screen "statistic" 800x480, template "Main"
   Rectangle "Rectangle_33" at 0,128 size 732x281
      Visibility <- "Vis_reset_stat"
   TextField "Text field_68" at 197,132 size 338x58; Text 'Новая партия.'
      Visibility <- "Vis_reset_stat"
   Button "Button_15" at 135,324 size 196x75; TextOff 'Продолжить'
      on Click: SetBit("T3V3W3_DB_Reset_statistic"); ResetBit("Vis_reset_stat")
      Visibility <- "Vis_reset_stat"
   Button "Button_6" at 391,323 size 196x75; TextOff 'Отмена'
      on Click: ResetBit("Vis_reset_stat")
      Visibility <- "Vis_reset_stat"
   TextField "Text field_69" at 200,186 size 333x46; Text 'Название партии:'
      Visibility <- "Vis_reset_stat"
   TextField "Text field_70" at 118,295 size 498x28; Text 'В партии может быть максимум 3000 коробок!'
      Visibility <- "Vis_reset_stat"
   IOField "I/O field_57" at 60,232 size 613x48; FormatPattern ?????????????????????????
      ProcessValue <- "T3V3W3_DB_LocalVar_name_part"
      Visibility <- "Vis_reset_stat"
   Button "Button_5" at 14,415 size 211x58; TextOff 'Обзор'
      on Click: ActivateScreen("Root screen", 0); SetTag("main_screens", 0)
      Appearance <- "main_screens"
   Button "Button_14" at 264,415 size 211x58; TextOff 'Вес'
      on Click: ActivateScreen("weight", 0); SetTag("main_screens", 1)
      Appearance <- "main_screens"
   Button "Button_7" at 513,415 size 211x58; TextOff 'Статистика'
      on Click: ActivateScreen("statistic", 0); SetTag("main_screens", 2); SetTag("stat_view", 0)
      Appearance <- "main_screens"
   Button "Button_8" at 150,363 size 211x46; TextOff 'Данные'
      on Click: ActivateScreen("statistic", 0); SetTag("stat_view", 0)
      Appearance <- "stat_view"
   Button "Button_9" at 372,363 size 211x46; TextOff 'Память'
      on Click: ActivateScreen("Memory", 0); SetTag("stat_view", 1)
      Appearance <- "stat_view"
   IOField "I/O field_1" at 122,58 size 57x22; FormatPattern 99.99
      ProcessValue <- "Statistic_DB_move_stat_Instance_box_weight{1}"
   TextField "Text field_1" at 122,0 size 231x23; Text 'Вес по коробкам в партии:'
   IOField "I/O field_2" at 153,29 size 47x22; FormatPattern 9999
      ProcessValue <- "b_1"
   TextField "Text field_2" at 122,29 size 43x23; Text '№'
   TextField "Text field_3" at 181,58 size 43x23; Text 'кг'
   IOField "I/O field_3" at 122,126 size 57x22; FormatPattern 99.99
      ProcessValue <- "Statistic_DB_move_stat_Instance_box_weight{6}"
   IOField "I/O field_4" at 153,96 size 47x22; FormatPattern 9999
      ProcessValue <- "b_6"
   TextField "Text field_4" at 122,96 size 43x23; Text '№'
   TextField "Text field_5" at 181,126 size 43x23; Text 'кг'
   IOField "I/O field_5" at 122,193 size 57x22; FormatPattern 99.99
      ProcessValue <- "Statistic_DB_move_stat_Instance_box_weight{11}"
   IOField "I/O field_6" at 153,164 size 47x22; FormatPattern 9999
      ProcessValue <- "b_11"
   TextField "Text field_6" at 122,164 size 43x23; Text '№'
   TextField "Text field_7" at 181,193 size 43x23; Text 'кг'
   IOField "I/O field_7" at 122,261 size 57x22; FormatPattern 99.99
      ProcessValue <- "Statistic_DB_move_stat_Instance_box_weight{16}"
   IOField "I/O field_8" at 153,231 size 47x22; FormatPattern 9999
      ProcessValue <- "b_16"
   TextField "Text field_8" at 122,231 size 43x23; Text '№'
   TextField "Text field_9" at 181,261 size 43x23; Text 'кг'
   IOField "I/O field_9" at 122,329 size 57x22; FormatPattern 99.99
      ProcessValue <- "Statistic_DB_move_stat_Instance_box_weight{21}"
   IOField "I/O field_10" at 153,299 size 47x22; FormatPattern 9999
      ProcessValue <- "b_21"
   TextField "Text field_10" at 122,299 size 43x23; Text '№'
   TextField "Text field_11" at 181,329 size 43x23; Text 'кг'
   IOField "I/O field_11" at 232,58 size 57x22; FormatPattern 99.99
      ProcessValue <- "Statistic_DB_move_stat_Instance_box_weight{2}"
   IOField "I/O field_12" at 263,29 size 47x22; FormatPattern 9999
      ProcessValue <- "b_2"
   TextField "Text field_12" at 232,29 size 43x23; Text '№'
   TextField "Text field_13" at 291,58 size 43x23; Text 'кг'
   IOField "I/O field_13" at 232,126 size 57x22; FormatPattern 99.99
      ProcessValue <- "Statistic_DB_move_stat_Instance_box_weight{7}"
   IOField "I/O field_14" at 263,96 size 47x22; FormatPattern 9999
      ProcessValue <- "b_7"
   TextField "Text field_14" at 232,96 size 43x23; Text '№'
   TextField "Text field_15" at 291,126 size 43x23; Text 'кг'
   IOField "I/O field_15" at 232,193 size 57x22; FormatPattern 99.99
      ProcessValue <- "Statistic_DB_move_stat_Instance_box_weight{12}"
   IOField "I/O field_16" at 263,164 size 47x22; FormatPattern 9999
      ProcessValue <- "b_12"
   TextField "Text field_16" at 232,164 size 43x23; Text '№'
   TextField "Text field_17" at 291,193 size 43x23; Text 'кг'
   IOField "I/O field_17" at 232,261 size 57x22; FormatPattern 99.99
      ProcessValue <- "Statistic_DB_move_stat_Instance_box_weight{17}"
   IOField "I/O field_18" at 263,231 size 47x22; FormatPattern 9999
      ProcessValue <- "b_17"
   TextField "Text field_18" at 232,231 size 43x23; Text '№'
   TextField "Text field_19" at 291,261 size 43x23; Text 'кг'
   IOField "I/O field_19" at 232,329 size 57x22; FormatPattern 99.99
      ProcessValue <- "Statistic_DB_move_stat_Instance_box_weight{22}"
   IOField "I/O field_20" at 263,299 size 47x22; FormatPattern 9999
      ProcessValue <- "b_22"
   TextField "Text field_20" at 232,299 size 43x23; Text '№'
   TextField "Text field_21" at 291,329 size 43x23; Text 'кг'
   IOField "I/O field_21" at 342,58 size 57x22; FormatPattern 99.99
      ProcessValue <- "Statistic_DB_move_stat_Instance_box_weight{3}"
   IOField "I/O field_22" at 373,29 size 47x22; FormatPattern 9999
      ProcessValue <- "b_3"
   TextField "Text field_22" at 342,29 size 43x23; Text '№'
   TextField "Text field_23" at 401,58 size 43x23; Text 'кг'
   IOField "I/O field_23" at 342,126 size 57x22; FormatPattern 99.99
      ProcessValue <- "Statistic_DB_move_stat_Instance_box_weight{8}"
   IOField "I/O field_24" at 373,96 size 47x22; FormatPattern 9999
      ProcessValue <- "b_8"
   TextField "Text field_24" at 342,96 size 43x23; Text '№'
   TextField "Text field_25" at 401,126 size 43x23; Text 'кг'
   IOField "I/O field_25" at 342,193 size 57x22; FormatPattern 99.99
      ProcessValue <- "Statistic_DB_move_stat_Instance_box_weight{13}"
   IOField "I/O field_26" at 373,164 size 47x22; FormatPattern 9999
      ProcessValue <- "b_13"
   TextField "Text field_26" at 342,164 size 43x23; Text '№'
   TextField "Text field_27" at 401,193 size 43x23; Text 'кг'
   IOField "I/O field_27" at 342,261 size 57x22; FormatPattern 99.99
      ProcessValue <- "Statistic_DB_move_stat_Instance_box_weight{18}"
   IOField "I/O field_28" at 373,231 size 47x22; FormatPattern 9999
      ProcessValue <- "b_18"
   TextField "Text field_28" at 342,231 size 43x23; Text '№'
   TextField "Text field_29" at 401,261 size 43x23; Text 'кг'
   IOField "I/O field_29" at 342,329 size 57x22; FormatPattern 99.99
      ProcessValue <- "Statistic_DB_move_stat_Instance_box_weight{23}"
   IOField "I/O field_30" at 373,299 size 47x22; FormatPattern 9999
      ProcessValue <- "b_23"
   TextField "Text field_30" at 342,299 size 43x23; Text '№'
   TextField "Text field_31" at 401,329 size 43x23; Text 'кг'
   IOField "I/O field_31" at 452,58 size 57x22; FormatPattern 99.99
      ProcessValue <- "Statistic_DB_move_stat_Instance_box_weight{4}"
   IOField "I/O field_32" at 483,29 size 47x22; FormatPattern 9999
      ProcessValue <- "b_4"
   TextField "Text field_32" at 452,29 size 43x23; Text '№'
   TextField "Text field_33" at 511,58 size 43x23; Text 'кг'
   IOField "I/O field_33" at 452,126 size 57x22; FormatPattern 99.99
      ProcessValue <- "Statistic_DB_move_stat_Instance_box_weight{9}"
   IOField "I/O field_34" at 483,96 size 47x22; FormatPattern 9999
      ProcessValue <- "b_9"
   TextField "Text field_34" at 452,96 size 43x23; Text '№'
   TextField "Text field_35" at 511,126 size 43x23; Text 'кг'
   IOField "I/O field_35" at 452,193 size 57x22; FormatPattern 99.99
      ProcessValue <- "Statistic_DB_move_stat_Instance_box_weight{14}"
   IOField "I/O field_36" at 483,164 size 47x22; FormatPattern 9999
      ProcessValue <- "b_14"
   TextField "Text field_36" at 452,164 size 43x23; Text '№'
   TextField "Text field_37" at 511,193 size 43x23; Text 'кг'
   IOField "I/O field_37" at 452,261 size 57x22; FormatPattern 99.99
      ProcessValue <- "Statistic_DB_move_stat_Instance_box_weight{19}"
   IOField "I/O field_38" at 483,231 size 47x22; FormatPattern 9999
      ProcessValue <- "b_19"
   TextField "Text field_38" at 452,231 size 43x23; Text '№'
   TextField "Text field_39" at 511,261 size 43x23; Text 'кг'
   IOField "I/O field_39" at 452,329 size 57x22; FormatPattern 99.99
      ProcessValue <- "Statistic_DB_move_stat_Instance_box_weight{24}"
   IOField "I/O field_40" at 483,299 size 47x22; FormatPattern 9999
      ProcessValue <- "b_24"
   TextField "Text field_40" at 452,299 size 43x23; Text '№'
   TextField "Text field_41" at 511,329 size 43x23; Text 'кг'
   IOField "I/O field_41" at 562,58 size 57x22; FormatPattern 99.99
      ProcessValue <- "Statistic_DB_move_stat_Instance_box_weight{5}"
   IOField "I/O field_42" at 593,29 size 47x22; FormatPattern 9999
      ProcessValue <- "b_5"
   TextField "Text field_42" at 562,29 size 43x23; Text '№'
   TextField "Text field_43" at 621,58 size 43x23; Text 'кг'
   IOField "I/O field_43" at 562,126 size 57x22; FormatPattern 99.99
      ProcessValue <- "Statistic_DB_move_stat_Instance_box_weight{10}"
   IOField "I/O field_44" at 593,96 size 47x22; FormatPattern 9999
      ProcessValue <- "b_10"
   TextField "Text field_44" at 562,96 size 43x23; Text '№'
   TextField "Text field_45" at 621,126 size 43x23; Text 'кг'
   IOField "I/O field_45" at 562,193 size 57x22; FormatPattern 99.99
      ProcessValue <- "Statistic_DB_move_stat_Instance_box_weight{15}"
   IOField "I/O field_46" at 593,164 size 47x22; FormatPattern 9999
      ProcessValue <- "b_15"
   TextField "Text field_46" at 562,164 size 43x23; Text '№'
   TextField "Text field_47" at 621,193 size 43x23; Text 'кг'
   IOField "I/O field_47" at 562,261 size 57x22; FormatPattern 99.99
      ProcessValue <- "Statistic_DB_move_stat_Instance_box_weight{20}"
   IOField "I/O field_48" at 593,231 size 47x22; FormatPattern 9999
      ProcessValue <- "b_20"
   TextField "Text field_48" at 562,231 size 43x23; Text '№'
   TextField "Text field_49" at 621,261 size 43x23; Text 'кг'
   IOField "I/O field_49" at 562,329 size 57x22; FormatPattern 99.99
      ProcessValue <- "Statistic_DB_move_stat_Instance_box_weight{25}"
   IOField "I/O field_50" at 593,299 size 47x22; FormatPattern 9999
      ProcessValue <- "b_25"
   TextField "Text field_50" at 562,299 size 43x23; Text '№'
   TextField "Text field_51" at 621,329 size 43x23; Text 'кг'
   GraphicView "Graphic view_1" at 664,24 size 57x50; Picture "u_grey"
   GraphicView "Graphic view_2" at 662,309 size 57x50; Picture "nope"
   TextField "Text field_52" at 22,21 size 72x23; Text 'Партия:'
   TextField "Text field_54" at 5,60 size 82x23; Text 'Коробок:'
   IOField "I/O field_52" at 36,78 size 47x22; FormatPattern 9999
      ProcessValue <- "T3V3W3_DB_Statistic_Count"
   TextField "Text field_55" at 81,78 size 43x23; Text 'шт'
   TextField "Text field_56" at 5,94 size 77x42; Text 'Средний вес:'
   IOField "I/O field_53" at 32,131 size 77x22; FormatPattern 99.99
      ProcessValue <- "T3V3W3_DB_Statistic_Mid_weight"
   TextField "Text field_57" at 81,131 size 43x23; Text 'кг'
   Button "Button_1" at 663,25 size 57x50; TextOff 'Text'
      on Click: SetBit("Statistic_DB_move_stat_Instance_up")
   Button "Button_2" at 663,309 size 57x50; TextOff 'Text'
      on Click: SetBit("Statistic_DB_move_stat_Instance_down")
   TextField "Text field_58" at 22,187 size 72x23; Text 'Партия:'
   TextField "Text field_59" at 17,205 size 82x23; Text 'Прошлая'
   TextField "Text field_60" at 9,228 size 82x23; Text 'Коробок:'
   IOField "I/O field_55" at 40,246 size 47x22; FormatPattern 9999
      ProcessValue <- "T3V3W3_DB_Statistic_Count_old"
   TextField "Text field_61" at 85,246 size 43x23; Text 'шт'
   TextField "Text field_62" at 9,259 size 77x42; Text 'Средний вес:'
   IOField "I/O field_56" at 35,296 size 54x22; FormatPattern 99.99
      ProcessValue <- "T3V3W3_DB_Statistic_Mid_weight_old"
   TextField "Text field_63" at 81,296 size 43x23; Text 'кг'
   TextField "Text field_53" at 6,38 size 104x23; Text 'Актуальная'
   Button "Button_3" at 658,165 size 69x52; TextOff 'Новая партия'
      on Click: SetBit("Vis_reset_stat")
      Visibility <- "Logic_DB_Start_weight"
   TextField "Text field_64" at 5,147 size 87x23; Text 'Общ. вес:'
   IOField "I/O field_51" at 8,165 size 77x22; FormatPattern 99999.9
      ProcessValue <- "T3V3W3_DB_Statistic_Weight"
   TextField "Text field_65" at 80,163 size 43x23; Text 'кг'
   TextField "Text field_66" at 9,313 size 87x23; Text 'Общ. вес:'
   IOField "I/O field_54" at 12,331 size 77x22; FormatPattern 99999.9
      ProcessValue <- "T3V3W3_DB_Statistic_Weight_old"
   TextField "Text field_67" at 84,329 size 43x23; Text 'кг'
   Button "Button_4" at 658,79 size 69x52; TextOff 'В начало'
      on Click: SetBit("Statistic_DB_move_stat_Instance_In_the_beggin")
   IOField "I/O field_58" at 352,1 size 313x22; FormatPattern ?????????????????????????
      ProcessValue <- "T3V3W3_DB_LocalVar_name_part"

Template "Main" 800x480
   Button "Button_1" at 735,5 size 60x60; TextOff 'Text'; PictureOff "home_2"
      on Click: ActivateScreen("Root screen", 0); SetTag("main_screens", 0)
   Button "Button_2" at 735,84 size 60x60; TextOff 'Text'; PictureOff "sett"
      on Click: ActivateScreen("SP", 0); SetTag("Sp_view", 1)
   Button "Button_4" at 735,163 size 60x60; TextOff 'Text'; PictureOff "sett_1"
      on Click: ActivateScreen("Monitor", 0); SetTag("settings", 0)
   Button "Button_5" at 735,242 size 60x60; TextOff 'Text'; PictureOff "home_1"; PictureList "Alarm"
      on Click: ActivateScreen("Alarms", 0)
      ProcessValue <- "Any_Alm"
   Button "Button_6" at 735,321 size 60x60; TextOff 'Text'; PictureOff "back"
      on Click: function_efd93a16()
   Button "Button_7" at 735,401 size 60x60; TextOff 'Text'; PictureOff "reset"
      on Click: SetBit("Reset_All")
   TextField "Template_Text field_1" at 735,63 size 60x15; Text 'F3'
   TextField "Template_Text field_2" at 735,222 size 60x15; Text 'F5'
   TextField "Template_Text field_3" at 735,143 size 60x15; Text 'F4'
   TextField "Template_Text field_4" at 735,300 size 60x15; Text 'F6'
   TextField "Template_Text field_5" at 735,460 size 60x15; Text 'F8'
   TextField "Template_Text field_6" at 735,380 size 60x15; Text 'F7'

screen "1.1_Recalibration" 800x480, template "Template_1"
   TextField "OBJECT_35" at 0,2 size 510x34; Text '1.1.1 Mit Gewichten Nachjustieren / 1.1 Recalibration / 1.1.1 Réétalonnage avec poids étalon / Calibration'
   Button "Exit to Service" at 45,390 size 80x80; TextOn 'Texte / text'; TextOff 'Texte / text'; PictureOff "Exit"
      on Release: ActivateScreen("Monitor", 0); SetTag("WP231PR_DB_CMD_A", 2034)
      on Press: SetTag("WP231PR_DB_s_CMD2_i_CMD_CODE", '2'); SetBit("WP231PR_DB_s_CMD2_bo_CMD_TRIGGER"); SetTag("WP231PR_DB_CMD_B", 0)
   Group "Group" at 700,5 size 95x30; Text 'Service'; PictureList "Signal_grey_yellow"
   Button "Up_to Setup_5_Min_01" at 545,390 size 80x80; TextOn 'Texte / text'; TextOff 'Texte / text'; PictureOff "Left"
      on Release: SetTag("WP231PR_DB_CMD_A", 2034)
      on Press: ActivateScreen("0.0.0_Service_Recalibration", 0); SetTag("WP231PR_DB_CMD_B", 0)
   IOField "OBJECT_301" at 0,41 size 800x90; FormatPattern ????????????????
      ProcessValue <- "WP231PR_DB_DR34_ASCII_DISPLAY"
   Button "OBJECT_28" at 110,133 size 580x70; TextOn 'Texte / text'; TextOff 'Justagegewicht 0 setzen / Set Calibration Weight 0 / Placez le poids étalon 0 / Acknowledge Empty Bin'
      on Press: SetTag("WP231PR_DB_s_CMD2_i_CMD_CODE", '60'); SetBit("WP231PR_DB_s_CMD2_bo_CMD_TRIGGER")
   Button "OBJECT_31" at 110,204 size 580x70; TextOn 'Texte / text'; TextOff 'Justagegewicht 1 setzen / Set Calibration Weight 1 / Placez le poids étalon 1 / Put & Acknowledge Calibration Weight'
      on Press: SetTag("WP231PR_DB_s_CMD2_i_CMD_CODE", '61'); SetBit("WP231PR_DB_s_CMD2_bo_CMD_TRIGGER")
   Button "OBJECT_3" at 110,276 size 580x70; TextOn 'Texte / text'; TextOff 'Justagegewicht 2 setzen (optional) / Set Calibration Weight 2 (optional) / Placez le poids étalon 2 (option) / Put & Acknowledge Calibration Weight'
      on Press: SetTag("WP231PR_DB_s_CMD2_i_CMD_CODE", '62'); SetBit("WP231PR_DB_s_CMD2_bo_CMD_TRIGGER")
   Button "Schaltfläche_1" at 670,390 size 80x80; TextOn 'Texte'; TextOff 'Texte'; PictureOff "Q_Mark"
      on Press: SetBit("S1_SHOW_HELP")
   TextField "OBJECT_4" at 210,352 size 207x32; Text 'Aktuelle Digits ADC: / Current ADC digits: / Valeur CAN / Error occurred'
      Visibility <- "S1_SHOW_HELP"
   IOField "I/O field_5" at 442,351 size 136x32; FormatPattern 9999999999
      ProcessValue <- "WP231PR_DB_DR31_DIGITS_FILTERED"
      Visibility <- "S1_SHOW_HELP"
   GraphicIOField "OBJECT_19" at 765,5 size 30x30; PictureList "Signal_grey_yellow"
      ProcessValue <- "WP231PR_DB_s_IO_DATA_SCALE_STATUS_2_SERVICE_MODE"
   TextField "OBJECT_37" at 700,7 size 57x25; Text 'Service / Error occurred'
   Rectangle "Rechteck_1" at 0,131 size 799x348
      Visibility <- "S1_SHOW_HELP"
   TextField "OBJECT_2" at 73,165 size 334x47; Text 'Justagegewicht 0: / Calibration weight 0: / Poids étalon 0: / Calibration'
      Visibility <- "S1_SHOW_HELP"
   TextField "OBJECT_1" at 73,230 size 334x47; Text 'Justagegewicht 1: / Calibration weight 1: / Poids étalon 1: / Calibration'
      Visibility <- "S1_SHOW_HELP"
   IOField "I/O field_1" at 415,230 size 166x47; FormatPattern 99999.99
      ProcessValue <- "WP231PR_DB_DR03_CALIB_WEIGHT_1"
      Visibility <- "S1_SHOW_HELP"
   IOField "I/O field_2" at 571,230 size 134x47; FormatPattern ????
      ProcessValue <- "WP231PR_DB_DR03_WEIGHT_UNIT"
      Visibility <- "S1_SHOW_HELP"
   IOField "I/O field_3" at 415,165 size 166x47; FormatPattern 99999.99
      ProcessValue <- "WP231PR_DB_DR03_CALIB_WEIGHT_0"
      Visibility <- "S1_SHOW_HELP"
   IOField "I/O field_4" at 571,165 size 134x47; FormatPattern ????
      ProcessValue <- "WP231PR_DB_DR03_WEIGHT_UNIT"
      Visibility <- "S1_SHOW_HELP"
   TextField "OBJECT_5" at 73,300 size 334x47; Text 'Justagegewicht 2: / Calibration weight 2: / Poids étalon 2: / Calibration'
      Visibility <- "S1_SHOW_HELP"
   IOField "I/O field_6" at 415,300 size 166x47; FormatPattern 99999.99
      ProcessValue <- "WP231PR_DB_DR03_CALIB_WEIGHT_2"
      Visibility <- "S1_SHOW_HELP"
   IOField "I/O field_7" at 571,300 size 134x47; FormatPattern ????
      ProcessValue <- "WP231PR_DB_DR03_WEIGHT_UNIT"
      Visibility <- "S1_SHOW_HELP"
   Button "Schaltfläche_2" at 642,420 size 150x50; TextOn 'Texte'; TextOff 'OK'
      on Press: ResetBit("S1_SHOW_HELP")
      Visibility <- "S1_SHOW_HELP"

screen "1.2.1_Quick_Start_1" 800x480, template "Template_1"
   TextField "OBJECT_33" at 0,0 size 440x34; Text '1.2.1 Quick Start 1 von 5 / 1.2.1 Quick Start 1 of 5 / 1.2.1 Mise en service rapide 1/5 / Setup 1/3'
   Button "Exit to Service" at 45,390 size 80x80; TextOn 'Texte / text'; TextOff 'Texte / text'; PictureOff "Exit"
      on Release: ActivateScreen("Monitor", 0)
      on Press: SetTag("WP231PR_DB_s_CMD2_i_CMD_CODE", '2'); SetBit("WP231PR_DB_s_CMD2_bo_CMD_TRIGGER")
   Button "Factory settings" at 110,112 size 580x90; TextOn 'Texte / text'; TextOff '"Quick Start" mit bestehenden Einstellungen / Run "Quick Start" with existing settings / Démarrage rapide avec les paramètres actuels / Acknowledge Empty Bin'
      on Release: ActivateScreen("1.2.2_Quick_Start_2", 0)
      on Press: SetTag("WP231PR_DB_s_CMD2_i_CMD_CODE", '2003'); SetBit("WP231PR_DB_s_CMD2_bo_CMD_TRIGGER")
   Group "Group" at 700,5 size 95x30; Text 'Service'; PictureList "Signal_grey_yellow"
   Button "Factory settings_1" at 110,237 size 580x90; TextOn 'Texte / text'; TextOff '"Quick Start" mit Werkseinstellungen / Run "Quick Start" with factory default settings / Démarrage rapide avec les paramètres usine / Acknowledge Empty Bin'
      on Release: ActivateScreen("1.2.2_Quick_Start_2", 0); SetTag("WP231PR_DB_s_CMD2_i_CMD_CODE", '2003'); SetBit("WP231PR_DB_s_CMD2_bo_CMD_TRIGGER")
      on Press: SetTag("WP231PR_DB_s_CMD1_i_CMD_CODE", 12); SetBit("WP231PR_DB_s_CMD1_bo_CMD_TRIGGER")
   Button "Schaltfläche_1" at 360,390 size 80x80; TextOn 'Texte'; TextOff 'Texte'; PictureOff "Q_Mark"
      on Press: SetBit("S1_SHOW_HELP")
   GraphicIOField "OBJECT_19" at 765,5 size 30x30; PictureList "Signal_grey_yellow"
      ProcessValue <- "WP231PR_DB_s_IO_DATA_SCALE_STATUS_2_SERVICE_MODE"
   TextField "OBJECT_37" at 700,7 size 57x25; Text 'Service / Error occurred'
   TextField "Textfeld_1" at 0,57 size 800x422; Text '"Quick Start" ermöglicht eine schnelle Basis-Inbetriebnahme der Waage. Es besteht die Möglichkeit die Waage mit oder ohne Justagegewichte zu justieren. "Quick Start" kann mit den bestehenden Waagenparametern, als auch mit geladenen Werkseinstellungen durchgeführt werden. "Quick Start" allows a fast and easy basic commissioning of the scale. It is possible to calibrate the scale with or without calibration weights. You can enter the "Quick Start" procedure with loaded factory settings or with maintaining the scale settings. Le démarrage rapide pour une mise en service en quelques minutes'
      Visibility <- "S1_SHOW_HELP"
   Button "Schaltfläche_2" at 643,423 size 150x50; TextOn 'Texte'; TextOff 'OK'
      on Press: ResetBit("S1_SHOW_HELP")
      Visibility <- "S1_SHOW_HELP"

screen "1.2.2_Quick_Start_2" 800x480, template "Template_1"
   TextField "OBJECT_33" at 0,0 size 440x34; Text '1.2.2 Quick Start 2 von 5 / 1.2.2 Quick Start 2 of 5 / 1.2.2 Mise en service rapide 2/5 / Setup 1/3'
   Button "Exit to Service" at 45,390 size 80x80; TextOn 'Texte / text'; TextOff 'Texte / text'; PictureOff "Exit"
      on Release: ActivateScreen("Monitor", 0)
      on Press: SetTag("WP231PR_DB_s_CMD2_i_CMD_CODE", '2'); SetBit("WP231PR_DB_s_CMD2_bo_CMD_TRIGGER")
   Group "Group" at 700,5 size 95x30; Text 'Service'; PictureList "Signal_grey_yellow"
   TextField "OBJECT_306" at 234,90 size 179x29; Text 'Waagenname / Scale Name / Nom de la balance / Scale name'
   IOField "OBJECT_307" at 420,84 size 172x40; HelpText 'Name der Waage (Produkt, Anlagenteil o.Ä.) / Nom de la balance'; FormatPattern ????????????
      ProcessValue <- "WP231PR_DB_DR03_SCALE_NAME"
   TextField "OBJECT_7" at 258,141 size 151x29; Text 'Gewichtseinheit / Weight unit / Unité poids / Weight Unit'
   IOField "OBJECT_28" at 420,134 size 172x40; HelpText 'Gewichtseinheit (z.B. g, kg oder t) / Unité poids (par ex. g, kg ou t)'; FormatPattern ????
      ProcessValue <- "WP231PR_DB_DR03_WEIGHT_UNIT"
   TextField "OBJECT_9" at 129,285 size 283x29; Text 'Minimaler Wägebereich (in d) / Minimum weight (in d) / Poids min (en d) / Weight Unit'
   TextField "OBJECT_10" at 159,330 size 254x29; Text 'Maximaler Wägebereich / Maximum weight / Plage maximale de pesage / Weight Unit'
   TextField "OBJECT_11" at 252,237 size 159x29; Text 'Ziffernschritt (d) / Resolution / Résolution (d) / Weight Unit'
   IOField "OBJECT_29" at 420,279 size 172x40; HelpText 'Bei geeichten Waagen mind. 20 x Ziffernschritt d. Bei nicht eichpflichtigen Waagen kann der minimale Wägebereich mit 0 definiert werden. / 20 x d pour usage certifié, sinon pas de limitation (0 par exemple)'; FormatPattern 999
      ProcessValue <- "WP231PR_DB_DR03_MIN_WEIGHT_D"
   IOField "OBJECT_12" at 420,325 size 173x40; HelpText 'Maximales Gewicht auf der Waage. Bei geeichten Waagen bitte entsprechende Einschränkungen beachten! / Poids max. sur la balance'; FormatPattern 9999999.9999
      ProcessValue <- "WP231PR_DB_DR03_MAX_WEIGHT"
   IOField "OBJECT_13" at 420,230 size 172x40; HelpText 'Ziffernschritt der Waage. Ist die Gewichts einheit "kg" bedeutet ein Ziffernschritt von 0,1 dass die Waage in 0,1kg Schritten auflöst. / Résolution de la balance. Avec un unité de poids de 1kg, la résolution de 0,1 signifie 0,1kg'; FormatPattern 9999.9999
      ProcessValue <- "WP231PR_DB_DR03_RESOLUTION_D"
   IOField "I/O field_2" at 596,325 size 60x40; FormatPattern ????
      ProcessValue <- "WP231PR_DB_DR03_WEIGHT_UNIT"
   TextField "Textfeld_1" at 609,283 size 18x29; Text 'x'
   Group "Group_1" at 607,242 size 62x59
   Button "Down to Setup_5_Min_03" at 690,390 size 80x80; TextOn 'Texte / text'; TextOff 'Texte / text'; PictureOff "Right"
      on Release: ActivateScreen("1.2.3_Quick_Start_3", 0)
   Button "Up_to Setup_5_Min_01" at 545,390 size 80x80; TextOn 'Texte / text'; TextOff 'Texte / text'; PictureOff "Left"
      on Release: ActivateScreen("1.2.1_Quick_Start_1", 0)
   TextField "OBJECT_6" at 8,188 size 403x29; Text 'Brutto-Kennung ("B" oder "G") / Indicator for Gross ("B" or "G") / Abréviation pour le poids brut ("B" ou "G") / Weight Unit'
   SymbolicIOField "Symbolic I/O field_1" at 421,187 size 172x31; TextOn '1'; TextOff '0'; TextList "003030_LETTER_FOR_GROSS_WEIGHT"
      ProcessValue <- "WP231PR_DB_DR03_LETTER_GROSS_WEIGHT_2"
   Button "Down to Setup_5_Min_1" at 360,390 size 80x80; TextOn 'Texte / text'; TextOff 'Texte / text'; PictureOff "Save"
      on Press: SetTag("WP231PR_DB_s_CMD2_i_CMD_CODE", '4003'); SetBit("WP231PR_DB_s_CMD2_bo_CMD_TRIGGER")
   GraphicIOField "OBJECT_19" at 765,5 size 30x30; PictureList "Signal_grey_yellow"
      ProcessValue <- "WP231PR_DB_s_IO_DATA_SCALE_STATUS_2_SIMULATION_MODE"
   TextField "OBJECT_37" at 700,7 size 57x25; Text 'Service / Error occurred'

screen "1.2.3_Quick_Start_3" 800x480, template "Template_1"
   TextField "OBJECT_35" at 0,0 size 440x34; Text '1.2.3 Quick Start 3 von 5 / 1.2.3 Quick Start 3 of 5 / 1.2.3 Mise en service rapide 3/5 / Quick Setup'
   Button "Exit to Service" at 45,390 size 80x80; TextOn 'Texte / text'; TextOff 'Texte / text'; PictureOff "Exit"
      on Release: ActivateScreen("Monitor", 0)
      on Press: SetTag("WP231PR_DB_s_CMD2_i_CMD_CODE", '2'); SetBit("WP231PR_DB_s_CMD2_bo_CMD_TRIGGER")
   TextField "OBJECT_38" at 34,80 size 762x32; Text 'Soll die Waage mit oder ohne Gewichte justiert werden? / Do you want to calibrate the scale with or without weights? / Calibration avec ou sans poids étalon? / For Quick Setup the scale must be empty'
   Button "Up_to Setup_5_Min_01" at 545,390 size 80x80; TextOn 'Texte / text'; TextOff 'Texte / text'; PictureOff "Left"
      on Release: ActivateScreen("1.2.2_Quick_Start_2", 0)
   Group "Group" at 700,5 size 95x30; Text 'Service'; PictureList "Signal_grey_yellow"
   Button "Factory settings" at 110,138 size 580x90; TextOn 'Texte / text'; TextOff 'Mit Gewichten justieren / Calibrate With Weights / Etalonner avec des poids étalons / Acknowledge Empty Bin'
      on Release: ActivateScreen("1.2.4_Quick_Start_Manual_Calibration_1", 0)
   Button "Factory settings_1" at 110,263 size 580x90; TextOn 'Texte / text'; TextOff 'Ohne Gewichte justieren (automatisch) Calibrate without weights (automatic) Calibration sans poids étalon Acknowledge Empty Bin'
      on Release: ActivateScreen("1.2.6_Quick_Start_4", 0)
      on Press: SetTag("WP231PR_DB_s_CMD2_i_CMD_CODE", '2010'); SetBit("WP231PR_DB_s_CMD2_bo_CMD_TRIGGER")
   Softkey "Softkey_F4" at -140,-147 size 0x0
      on KeyDown: ActivateScreen("1.2.6_Quick_Start_4", 0)
   GraphicIOField "OBJECT_19" at 765,5 size 30x30; PictureList "Signal_grey_yellow"
      ProcessValue <- "WP231PR_DB_s_IO_DATA_SCALE_STATUS_2_SERVICE_MODE"
   TextField "OBJECT_37" at 700,7 size 57x25; Text 'Service / Error occurred'
   TextField "Textfeld_1" at 0,57 size 800x422; Text 'Justage mit Gewichten: Es müssen mindestens 5% der Nennlast der Waage als Justagegewicht zur Verfügung stehen. Beispiel: 3 x 2t Wägezellen = 6t Nennlast --> Die Waage muss mit mindestens 300kg (5% von 6t) justiert werden. Wird der Justagepunkt 2 ebenfalls genutzt, muss dieser wiederum mindestens 300kg vom Justagepunkt 1 entfernt sein. Automatische Justage: Es sind keine Justagegewichte notwendig. Die Wägezellendaten müssen zur Verfügung stehen. Mechanische Einflüsse werden nicht berücksichtigt! Etalonnage avec un poids étalon. Au min 5% de la charge nominale des pesons'
      Visibility <- "S1_SHOW_HELP"
   Button "Schaltfläche_2" at 643,423 size 150x50; TextOn 'Texte'; TextOff 'OK'
      on Press: ResetBit("S1_SHOW_HELP")
      Visibility <- "S1_SHOW_HELP"

screen "1.2.4_Quick_Start_Manual_Calibration_1" 800x480, template "Template_1"
   TextField "OBJECT_33" at 0,0 size 630x34; Text '1.2.4 Quick Start - Justagegewichte 4 von 5 / 1.2.4 Quick Start - Calibration Weights 4 of 5 / 1.2.4 Mise en service rapide poids étalon 4/5 / Setup 1/3'
   TextField "OBJECT_306" at 157,135 size 206x32; Text 'Justagegewicht 0 / Calibration weight 0 / Poids étalon 0 / Scale name'
   Button "OBJECT_34" at 670,390 size 80x80; TextOn 'Texte / text'; TextOff 'Texte / text'; PictureOff "Right"
      on Release: ActivateScreen("1.2.5_Quick_Start_Manual_Calibration_2", 0); SetTag("WP231PR_DB_CMD_A", 2034)
      on Press: SetTag("WP231PR_DB_CMD_B", 2031)
   IOField "OBJECT_307" at 373,126 size 300x50; HelpText 'Falls die Waage zum Zeitpunkt der Justage nicht leer ist, kann das bekannte Gewicht in der Waage als "Justagegewicht 0" vorgegeben werden. / If the scale is not empty before adjusting, the known material weight in the scale can be defined as "Calibration weight 0". / Si pour l'étalonnage la balance n'est pas vide, il est possible d'utiliser le poids actuel comme poids étalon'; FormatPattern 999999.999
      ProcessValue <- "WP231PR_DB_DR03_CALIB_WEIGHT_0"
   TextField "OBJECT_7" at 158,192 size 206x32; Text 'Justagegewicht 1 / Calibration weight 1 / Poids étalon 1 / Weight Unit'
   IOField "OBJECT_28" at 373,182 size 300x50; HelpText 'Das "Justagegewicht 1" muss mindestens 5% der Nennlast der Waage entsprechen! / Le poids étalon doit être supérieur à 5% de la charge max des pesons'; FormatPattern 999999.999
      ProcessValue <- "WP231PR_DB_DR03_CALIB_WEIGHT_1"
   Button "OBJECT_24" at 45,390 size 80x80; TextOn 'Texte / text'; TextOff 'Texte / text'; PictureOff "Exit"
      on Release: ActivateScreen("Monitor", 0)
      on Press: SetTag("WP231PR_DB_s_CMD2_i_CMD_CODE", '2'); SetBit("WP231PR_DB_s_CMD2_bo_CMD_TRIGGER")
   TextField "OBJECT_6" at 42,248 size 320x32; Text 'Justagegewicht 2 (optional) / Calibration weight 2 (optional) / Poids étalon 2 (option) / Weight Unit'
   IOField "OBJECT_8" at 372,240 size 302x50; HelpText 'Mit "Justagegewicht 2" kann ein dritter Justagepunkt gesetzt werden. Es ist nicht zwingend erforderlich diesen zu setzen! Falls genutzt, muss der Abstand zwischen "Justagegewicht 1" und "Justagegewicht 2" mind. 5% der Nennlast der Waage entsprechen. Le poids étalon 2 permet d'avoir un troisième points d'étalonnage'; FormatPattern 999999.999
      ProcessValue <- "WP231PR_DB_DR03_CALIB_WEIGHT_2"
   IOField "I/O field_2" at 676,131 size 60x40; FormatPattern ????
      ProcessValue <- "WP231PR_DB_DR03_WEIGHT_UNIT"
   IOField "I/O field_1" at 676,189 size 60x40; FormatPattern ????
      ProcessValue <- "WP231PR_DB_DR03_WEIGHT_UNIT"
   IOField "I/O field_3" at 677,244 size 60x40; FormatPattern ????
      ProcessValue <- "WP231PR_DB_DR03_WEIGHT_UNIT"
   Group "Group" at 700,5 size 95x30; Text 'Service'; PictureList "Signal_grey_yellow"
   Button "Up_to Setup_5_Min_01" at 545,390 size 80x80; TextOn 'Texte / text'; TextOff 'Texte / text'; PictureOff "Left"
      on Release: ActivateScreen("1.2.3_Quick_Start_3", 0)
   Button "Schaltfläche_1" at 213,390 size 80x80; TextOn 'Texte'; TextOff 'Texte'; PictureOff "Q_Mark"
      on Press: SetBit("S1_SHOW_HELP")
   Button "OBJECT_1" at 360,390 size 80x80; TextOn 'Texte / text'; TextOff 'Texte / text'; PictureOff "Save"
      on Press: SetTag("WP231PR_DB_s_CMD2_i_CMD_CODE", '4003'); SetBit("WP231PR_DB_s_CMD2_bo_CMD_TRIGGER")
   GraphicIOField "OBJECT_19" at 765,5 size 30x30; PictureList "Signal_grey_yellow"
      ProcessValue <- "WP231PR_DB_s_IO_DATA_SCALE_STATUS_2_SIMULATION_MODE"
   TextField "OBJECT_37" at 700,7 size 57x25; Text 'Service / Error occurred'
   GraphicView "Grafikanzeige_1" at 4,7 size 793x470; Picture "char_curve"
      Visibility <- "S1_SHOW_HELP"
   Button "Schaltfläche_2" at 19,420 size 150x50; TextOn 'Texte'; TextOff 'OK'
      on Press: ResetBit("S1_SHOW_HELP")
      Visibility <- "S1_SHOW_HELP"

screen "1.2.5_Quick_Start_Manual_Calibration_2" 800x480, template "Template_1"
   TextField "OBJECT_35" at 0,0 size 691x34; Text '1.2.5 Quick Start - Justage mit Gewichten 5 von 5 / 1.2.5 Quick Start - Calibration with Weights / 1.2.5 Mise en service rapide poids étalon 5/5 / Calibration'
   IOField "OBJECT_301" at 0,41 size 800x90; FormatPattern ????????????????
      ProcessValue <- "WP231PR_DB_DR34_ASCII_DISPLAY"
   Group "Group" at 700,5 size 95x30; Text 'Service'; PictureList "Signal_grey_yellow"
   Button "Up_to Setup_5_Min_01" at 545,390 size 80x80; TextOn 'Texte / text'; TextOff 'Texte / text'; PictureOff "Left"
      on Release: ActivateScreen("1.2.4_Quick_Start_Manual_Calibration_1", 0); SetTag("WP231PR_DB_CMD_A", 2034)
      on Press: SetTag("WP231PR_DB_s_CMD2_i_CMD_CODE", '2003'); SetBit("WP231PR_DB_s_CMD2_bo_CMD_TRIGGER"); SetTag("WP231PR_DB_CMD_B", 0)
   Button "Exit to Service" at 45,390 size 80x80; TextOn 'Texte / text'; TextOff 'Texte / text'; PictureOff "Exit"
      on Release: ActivateScreen("Monitor", 0); SetTag("WP231PR_DB_CMD_A", 2034); SetTag("WP231PR_DB_s_CMD1_i_CMD_CODE", '2'); SetBit("WP231PR_DB_s_CMD1_bo_CMD_TRIGGER")
      on Press: SetTag("WP231PR_DB_s_CMD2_i_CMD_CODE", '2'); SetBit("WP231PR_DB_s_CMD2_bo_CMD_TRIGGER"); SetTag("WP231PR_DB_CMD_B", 0)
   Button "OBJECT_28" at 110,135 size 580x70; TextOn 'Texte / text'; TextOff 'Justagegewicht 0 setzen / Set Calibration Weight 0 / Placez le poids étalon 0 / Acknowledge Empty Bin'
      on Press: SetTag("WP231PR_DB_s_CMD2_i_CMD_CODE", '60'); SetBit("WP231PR_DB_s_CMD2_bo_CMD_TRIGGER")
   Button "OBJECT_31" at 110,207 size 580x70; TextOn 'Texte / text'; TextOff 'Justagegewicht 1 setzen / Set Calibration Weight 1 / Placez le poids étalon 1 / Put & Acknowledge Calibration Weight'
      on Press: SetTag("WP231PR_DB_s_CMD2_i_CMD_CODE", '61'); SetBit("WP231PR_DB_s_CMD2_bo_CMD_TRIGGER")
   Button "OBJECT_3" at 110,279 size 580x70; TextOn 'Texte / text'; TextOff 'Justagegewicht 2 setzen (optional) / Set Calibration Weight 2 (optional) / Placez le poids étalon 2 (option) / Put & Acknowledge Calibration Weight'
      on Press: SetTag("WP231PR_DB_s_CMD2_i_CMD_CODE", '62'); SetBit("WP231PR_DB_s_CMD2_bo_CMD_TRIGGER")
   GraphicIOField "OBJECT_19" at 765,5 size 30x30; PictureList "Signal_grey_yellow"
      ProcessValue <- "WP231PR_DB_s_IO_DATA_SCALE_STATUS_2_SIMULATION_MODE"
   TextField "OBJECT_37" at 700,7 size 57x25; Text 'Service / Error occurred'
   TextField "OBJECT_4" at 227,352 size 207x32; Text 'Aktuelle Digits ADC: / Current ADC digits: / Valeur CAN / Error occurred'
   IOField "I/O field_5" at 442,352 size 136x32; FormatPattern 9999999999
      ProcessValue <- "WP231PR_DB_DR31_DIGITS_FILTERED"

screen "1.2.6_Quick_Start_4" 800x480, template "Template_1"
   TextField "OBJECT_33" at 0,0 size 662x34; Text '1.2.6 Quick Start 4 von 5 / 1.2.6 Quick Start 4 of 5 - Load Cells Parameters / 1.2.6 Mise en service rapide 4/5 / Setup 1/3'
   Button "Down to Setup_5_Min_03" at 670,390 size 80x80; TextOn 'Texte / text'; TextOff 'Texte / text'; PictureOff "Right"
      on Release: ActivateScreen("1.2.7_Quick_Start_Automatic_Calibration", 0)
      on Press: SetTag("WP231PR_DB_CMD_A", 2034)
   TextField "OBJECT_7" at 297,150 size 264x32; Text 'Anzahl Auflagepunkte / Number of support points / Nombre de points d'appui / Weight Unit'
   IOField "OBJECT_28" at 580,142 size 130x45; HelpText 'Bei Silo mit drei Beinen = 3 Bei Silo mit vier Beinen = 4 usw. Hopper with 3 legs = 3 Hopper with 4 legs = 4 ASO. 3 pour un silo avec 3 pieds, 4 pour un silo à 4 pieds etc.'; FormatPattern 9
      ProcessValue <- "WP231PR_DB_DR10_NO_POINTS_OF_SUPPORT"
   Button "Exit to Service" at 45,390 size 80x80; TextOn 'Texte / text'; TextOff 'Texte / text'; PictureOff "Exit"
      on Release: ActivateScreen("Monitor", 0)
      on Press: SetTag("WP231PR_DB_s_CMD2_i_CMD_CODE", '2'); SetBit("WP231PR_DB_s_CMD2_bo_CMD_TRIGGER")
   TextField "OBJECT_308" at 201,259 size 358x32; Text 'Nennlast einer Wägezelle / Nominal load of one single load cell / Charge nominale d'un peson / Limit Freq. Low Pass Filter'
   TextField "OBJECT_9" at 39,206 size 528x32; Text 'Durchschnittskennwert aller Wägezellen (mV/V) / Average of all characteristic values (mV/V) / Valeur moyenne de la sensibilité des pesons (mV/V) / Stand Still Time'
   IOField "OBJECT_32" at 580,198 size 130x45; HelpText 'Kennwert Zelle 1 = 1,998 mV/V Kennwert Zelle 2 = 2,002 mV/V Kennwert Zelle 3 = 2,000 mV/V ======================== Durchschnitt = 2,000 mV/V Charact. Value Cell 1 = 1,998 mV/V Charact. Value Cell 2 = 2,002 mV/V Charact. Value Cell 3 = 2,000 mV/V =========================== Average = 2,000 mV/V Sensibilité peson 1 = 1,998 mV/V Sensibilité peson 2 = 2,002 mV/V Sensibilité peson 3 = 2,000 mV/V ======================== Moyenne = 2,000 mV/V'; FormatPattern 99.999999
      ProcessValue <- "WP231PR_DB_DR10_GAIN_LOAD_CELL"
   IOField "OBJECT_2" at 580,252 size 130x45; FormatPattern 999999999.9
      ProcessValue <- "WP231PR_DB_DR10_NOM_LOAD_ONE_LOAD_CELL"
   Button "Up_to Setup_5_Min_01" at 545,390 size 80x80; TextOn 'Texte / text'; TextOff 'Texte / text'; PictureOff "Left"
      on Release: ActivateScreen("1.2.3_Quick_Start_3", 0)
   IOField "I/O field_2" at 713,261 size 82x29; FormatPattern ????
      ProcessValue <- "WP231PR_DB_DR03_WEIGHT_UNIT"
   Group "Group" at 700,5 size 95x30; Text 'Service'; PictureList "Signal_grey_yellow"
   Button "Down to Setup_5_Min_1" at 360,390 size 80x80; TextOn 'Texte / text'; TextOff 'Texte / text'; PictureOff "Save"
      on Press: SetTag("WP231PR_DB_s_CMD1_i_CMD_CODE", 4010); SetBit("WP231PR_DB_s_CMD1_bo_CMD_TRIGGER")
   Softkey "Softkey_F4" at -140,-147 size 0x0
      on KeyDown: ActivateScreen("1.2.1_Quick_Start_1", 0)
   GraphicIOField "OBJECT_19" at 765,5 size 30x30; PictureList "Signal_grey_yellow"
      ProcessValue <- "WP231PR_DB_s_IO_DATA_SCALE_STATUS_2_SERVICE_MODE"
   TextField "OBJECT_37" at 700,7 size 57x25; Text 'Service / Error occurred'

screen "1.2.7_Quick_Start_Automatic_Calibration" 800x480, template "Template_1"
   TextField "OBJECT_35" at 0,0 size 679x34; Text '1.2.7 Quick Start - Automatische Justage 5 von 5 / 1.2.7 Quick Start - Automatic Calibration 5 of 5 / 1.2.7 Mise en service rapide étalonnage auto 5/5 / Quick Setup'
   Button "Exit to Service" at 45,390 size 80x80; TextOn 'Texte / text'; TextOff 'Texte / text'; PictureOff "Exit"
      on Release: ActivateScreen("Monitor", 0); SetTag("WP231PR_DB_CMD_A", 2034)
      on Press: SetTag("WP231PR_DB_s_CMD2_i_CMD_CODE", '2'); SetBit("WP231PR_DB_s_CMD2_bo_CMD_TRIGGER")
   TextField "OBJECT_38" at 72,181 size 718x29; Text 'Für die automatische Justage muss die Waage jetzt leer sein ! / For automatic calibration the scale needs to be empty now! / La balance doit être vide pour l'étalonnage automatique / For Quick Setup the scale must be empty'
   Button "Confirm_scale_empty" at 110,236 size 580x70; TextOn 'Texte / text'; TextOff 'Automatische Justage durchführen / Start Automatic Calibration / Effectue l'étalonnage automatique / Acknowledge Empty Bin'
      on Release: SetTag("WP231PR_DB_s_CMD2_i_CMD_CODE", '2003'); SetBit("WP231PR_DB_s_CMD2_bo_CMD_TRIGGER")
      on Press: SetTag("WP231PR_DB_s_CMD1_i_CMD_CODE", '82'); SetBit("WP231PR_DB_s_CMD1_bo_CMD_TRIGGER")
   Button "Up_to Setup_5_Min_01" at 545,390 size 80x80; TextOn 'Texte / text'; TextOff 'Texte / text'; PictureOff "Left"
      on Release: ActivateScreen("1.2.6_Quick_Start_4", 0)
   Group "Group" at 700,5 size 95x30; Text 'Service'; PictureList "Signal_grey_yellow"
   IOField "OBJECT_301" at 0,74 size 800x86; FormatPattern ????????????????
      ProcessValue <- "WP231PR_DB_DR34_ASCII_DISPLAY"
   Softkey "Softkey_F4" at -140,-147 size 0x0
      on KeyDown: ActivateScreen("1.2.6_Quick_Start_4", 0)
   GraphicIOField "OBJECT_19" at 765,5 size 30x30; PictureList "Signal_grey_yellow"
      ProcessValue <- "WP231PR_DB_s_IO_DATA_SCALE_STATUS_2_SIMULATION_MODE"
   TextField "OBJECT_37" at 700,7 size 57x25; Text 'Service / Error occurred'

screen "0.0.0_Service_Quick_Start" 800x480, template "Template_1"
   TextField "OBJECT_35" at 0,0 size 314x34; Text 'Quick Start - Warnung / Quick Start - Warning / Mise en service rapide / Calibration'
   Button "OBJECT_24" at 45,390 size 80x80; TextOn 'Texte / text'; TextOff 'Texte / text'; PictureOff "Exit"
      on Release: ActivateScreen("Monitor", 0)
      on Press: SetTag("WP231PR_DB_s_CMD2_i_CMD_CODE", 2); SetBit("WP231PR_DB_s_CMD2_bo_CMD_TRIGGER")
   TextField "OBJECT_1" at 24,89 size 127x33; Text 'Achtung! / Warning! / Attention / Calibration'
   TextField "OBJECT_2" at 20,119 size 773x120; Text 'Für "Quick Start" muss die Waage in den Service-Betrieb geschaltet werden. Sie haben Zugriff auf alle Waagenparameter! Der "Hilfe" Button der Touch-Tastatur beschreibt die Parameter. For "Quick Start" the scale needs to be in Serivce Mode. You will have full access to critical parameters! The "Help" button on the Touch-Keypad describes the single parameters. Mode service requis pour la mise en service rapide Calibration'
   Button "OBJECT_34" at 670,390 size 80x80; TextOn 'Texte / text'; TextOff 'Texte / text'; PictureOff "Right"
      on Release: ActivateScreen("1.2.1_Quick_Start_1", 0)
   Button "Service on_1" at 225,280 size 350x90; TextOn 'Texte / text'; TextOff 'Servicebetrieb einschalten Switch On "Service Mode" Mettre en mode service Acknowledge Empty Bin'
      on Press: SetTag("WP231PR_DB_s_CMD2_i_CMD_CODE", '1'); SetBit("WP231PR_DB_s_CMD2_bo_CMD_TRIGGER")
   Group "Group" at 700,5 size 95x30; Text 'Service'; PictureList "Signal_grey_yellow"
   Button "Zero" at 360,390 size 80x80; TextOn 'Texte / text'; TextOff '- 0 - / Menu'; PictureOff "Zero"
      on Release: SetTag("WP231PR_DB_s_CMD2_i_CMD_CODE", 1001); SetBit("WP231PR_DB_s_CMD2_bo_CMD_TRIGGER")
   GraphicIOField "OBJECT_19" at 765,5 size 30x30; PictureList "Signal_grey_yellow"
      ProcessValue <- "WP231PR_DB_s_IO_DATA_SCALE_STATUS_2_SERVICE_MODE"
   TextField "OBJECT_37" at 700,7 size 57x25; Text 'Service / Error occurred'

screen "0.0.0_Service_Recalibration" 800x480, template "Template_1"
   TextField "OBJECT_35" at 0,0 size 336x34; Text 'Nachjustage - Warnung / Recalibration - Warning / Réétalonnage / Calibration'
   Button "OBJECT_24" at 45,390 size 80x80; TextOn 'Texte / text'; TextOff 'Texte / text'; PictureOff "Exit"
      on Release: ActivateScreen("Monitor", 0)
      on Press: SetTag("WP231PR_DB_s_CMD2_i_CMD_CODE", 2); SetBit("WP231PR_DB_s_CMD2_bo_CMD_TRIGGER")
   TextField "OBJECT_1" at 24,89 size 127x33; Text 'Achtung! / Warning! / Attention / Calibration'
   TextField "OBJECT_2" at 18,130 size 767x91; Text 'Für die Nachjustage muss die Waage in den Service-Betrieb geschaltet werden. Sie haben Zugriff auf alle Waagenparameter. Die aktuelle Waagenkennlinie wird überschrieben! For "Recalibration" the scale needs to be in Service Mode. You will have full access to critical parameters! The current scale curve will be overwritten! Mode service requis pour le réétalonnage Calibration'
   Button "OBJECT_34" at 670,390 size 80x80; TextOn 'Texte / text'; TextOff 'Texte / text'; PictureOff "Right"
      on Release: ActivateScreen("1.1_Recalibration", 0); SetTag("WP231PR_DB_CMD_B", 2031)
      on Press: SetTag("WP231PR_DB_s_CMD2_i_CMD_CODE", '2003'); SetTag("WP231PR_DB_s_CMD2_bo_CMD_TRIGGER", 1)
   Button "Service on_1" at 225,280 size 350x90; TextOn 'Texte / text'; TextOff 'Servicebetrieb einschalten Switch On "Service Mode" Mettre en mode service Acknowledge Empty Bin'
      on Press: SetTag("WP231PR_DB_s_CMD2_i_CMD_CODE", '1'); SetBit("WP231PR_DB_s_CMD2_bo_CMD_TRIGGER")
   Group "Group" at 700,5 size 95x30; Text 'Service'; PictureList "Signal_grey_yellow"
   Button "Zero" at 360,390 size 80x80; TextOn 'Texte / text'; TextOff '- 0 - / Menu'; PictureOff "Zero"
      on Release: SetTag("WP231PR_DB_s_CMD2_i_CMD_CODE", 1001); SetBit("WP231PR_DB_s_CMD2_bo_CMD_TRIGGER")
   GraphicIOField "OBJECT_19" at 765,5 size 30x30; PictureList "Signal_grey_yellow"
      ProcessValue <- "WP231PR_DB_s_IO_DATA_SCALE_STATUS_2_SERVICE_MODE"
   TextField "OBJECT_37" at 700,7 size 57x25; Text 'Service / Error occurred'
*)